TYPE AX5000_P_0555 :
STRUCT
	Position_command_value_monitoring_window:UINT;
END_STRUCT
END_TYPE

(* stored: Version 1.1.0.1, ProductVersion 3.1.4024.3
   DUT AX5000_P_0555: Id {b5ee175a-acad-4a5a-b855-9891bf2f383e} *)
